/// This is the **Base** FB for every single FB
/// Inherited by:
FUNCTION_BLOCK FB_Test1_Base //< [FB_Test1](xref:ZK_Doc1.FB_Test1)
VAR_INPUT
	/// This is the first ___Input___
	/// Now comes a code example:
	/// ~~We dont need this~~
	/// ```st
	/// METHOD Method1
	/// VAR_INPUT
  	/// input1 : BOOL; //< what does this input do
  	///
  	/// /// or this one?
  	/// input2 : INT;
	/// END_VAR
	/// ```
	nInput1 : INT := 1; 
END_VAR
VAR_OUTPUT
	sOutput1 : T_MaxString := "This is output 1";
END_VAR
VAR
	nVar1 : INT;
	nVar2 : INT;
	sVar3 : T_MaxString;
	bVar4 : BOOL;
END_VAR
VAR CONSTANT
	nConst1 : INT := 2026;
	sConst2 : STRING(155) := 'Constant 2';
END_VAR
VAR PERSISTENT
	nVarPers : LREAL := 155.155;
	
END_VAR

METHOD INTERNAL M_SetVar : BOOL
VAR_INPUT
	nVarIn1 : INT;
END_VAR
P_nVar1 := nVarIn1;
M_SetVar := nVarIn1 >= 100;
RETURN;
END_METHOD

PROPERTY PRIVATE P_FOO : BOOL
GET
P_FOO := TRUE;
RETURN;
END_GET
SET
bVar4 := P_FOO;
END_SET
END_PROPERTY

PROPERTY PROTECTED P_nVar1 : INT
GET
P_nVar1 := nVar1;
RETURN;
END_GET
SET
nVar1 := P_nVar1;
END_SET
END_PROPERTY

END_FUNCTION_BLOCK

(* stored: Version 1.1.0.1
   POU FB_Test1_Base: Id {e8068e8a-7f86-46dd-bec1-e6051adfee17}, SpecialFunc None
   Method M_SetVar: Id {28b55f5b-b6d8-46c8-8db0-4904c22c755d}
   Property P_FOO: Id {e026ea42-fac1-4645-af70-a9e901d5f489}
   Get Get: Id {240f3e9c-8891-4b84-9b3c-8fdc3ea3faa5}
   Set Set: Id {3972200d-09a7-419a-9fa3-b190210b07b7}
   Property P_nVar1: Id {82e8eb42-a4dd-4381-bb3e-dd79da27e399}
   Get Get: Id {563656eb-c7e1-43af-b47e-7ee8483b1e45}
   Set Set: Id {fd64a189-af5a-4e05-ab98-256aac99ac1d} *)
